SUBAPPLICATION Toggle_RPC_FROM_Remote_QXA_OPC (* Geraet B (Station 12, 192.168.1.12): empfaengt den Trigger-Methodenaufruf von Geraet A per SERVER_0 (reiner RPC-Trigger, kein Wertwechsel-Trick, keine Bridge noetig), taktet die echte Toggle-Flipflop-Logik (AX_T_FF), schaltet DigitalOutput_Q1 und schreibt den neuen Zustand aktiv per CLIENT_1_0 zurueck auf Geraet A - 'SUB style': das Protokoll steckt im MyLib::sys-Composite, nicht in der Resource des Geraets *)
  (* Standard: 61499-2; Description: Copyright (c) 2026 Meisterschulen am Ostbahnhof This program and the accompanying materials are made available under the terms of the Eclipse Public License 2.0 which is available at https://www.eclipse.org/legal/epl-2.0/ SPDX-License-Identifier: EPL-2.0 *)
  (* Version 1.1, 2026-09-09, Franz Höpfinger, Meisterschulen am Ostbahnhof, Fix: TRIGGER_SERVER.RSP war nie verdrahtet - blockierte den OPC-UA-Server-Thread bis zu 4s (haelt open62541s globalen serviceMutex), verzoegerte dadurch JEDE OPC-UA-Statusmeldung projektweit. IND->RSP direkt verdrahtet. Siehe OPC_UA_VERNETZUNG.md Punkt 12. *)
  (* Version 1.0, 2026-09-02, Franz Höpfinger, Meisterschulen am Ostbahnhof, initial API and implementation and/or initial documentation *)
  PACKAGE MyLib::sys;
  IMPORT logiBUS::io::DQ::logiBUS_DO;
  IMPORT logiBUS::io::DQ::logiBUS_DO_S;
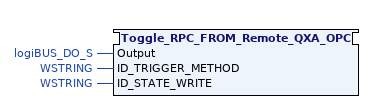
  VAR_INPUT
    Output : logiBUS::io::DQ::logiBUS_DO_S := logiBUS_DO::Invalid; (* Identify the Output Output_Q1..Q8 *)
    ID_TRIGGER_METHOD : WSTRING; (* Lokale Methodenadresse (ACTION=CREATE_METHOD) fuer den argumentlosen Trigger-Methodenaufruf, wird von Geraet A per CALL_METHOD aufgerufen *)
    ID_STATE_WRITE : WSTRING; (* Remote-Ziel-Adresse (BOOL, ACTION=WRITE) fuer den Flipflop-Zustand auf Geraet A *)
  END_VAR
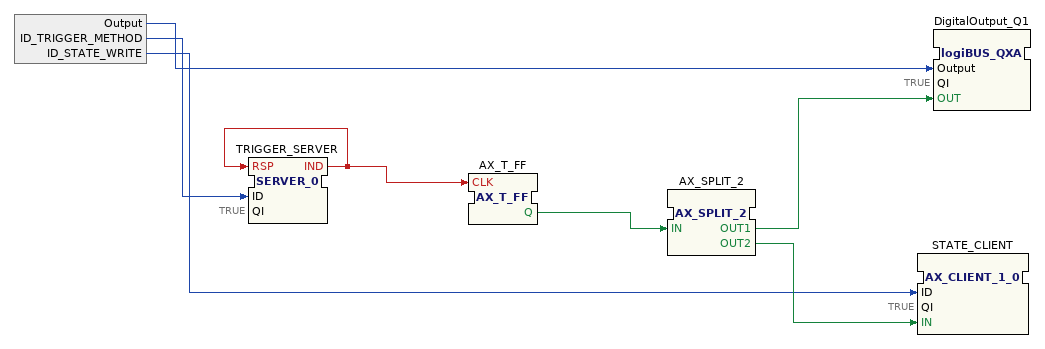
  FBS
    TRIGGER_SERVER : iec61499::net::SERVER_0(QI := TRUE);
    AX_T_FF : adapter::events::unidirectional::AX_T_FF;
    AX_SPLIT_2 : adapter::events::unidirectional::AX_SPLIT_2;
    DigitalOutput_Q1 : logiBUS::io::DQ::logiBUS_QXA(QI := TRUE);
    STATE_CLIENT : adapter::net::AX_CLIENT_1_0(QI := TRUE);
  END_FBS
  EVENT_CONNECTIONS
    TRIGGER_SERVER.IND TO AX_T_FF.CLK;
    TRIGGER_SERVER.IND TO TRIGGER_SERVER.RSP;
  END_CONNECTIONS
  DATA_CONNECTIONS
    Output TO DigitalOutput_Q1.Output;
    ID_TRIGGER_METHOD TO TRIGGER_SERVER.ID;
    ID_STATE_WRITE TO STATE_CLIENT.ID;
  END_CONNECTIONS
  ADAPTER_CONNECTIONS
    AX_T_FF.Q TO AX_SPLIT_2.IN;
    AX_SPLIT_2.OUT1 TO DigitalOutput_Q1.OUT;
    AX_SPLIT_2.OUT2 TO STATE_CLIENT.IN;
  END_CONNECTIONS
END_SUBAPPLICATION
